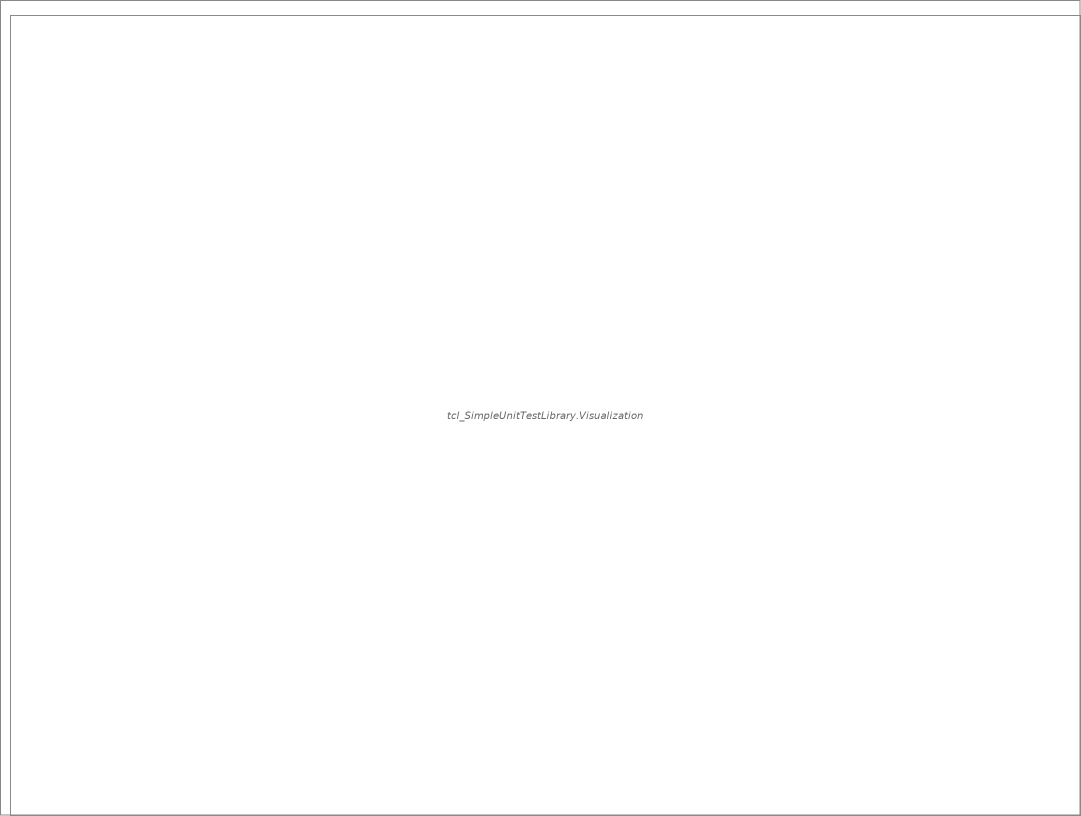
VISUALIZATION Visualization  // 1081x816
    Frame (10,15 1071x801)
        shows tcl_SimpleUnitTestLibrary.Visualization(TestRunner := PB_TestRunner.TestRunner)
END_VISUALIZATION

(* stored: Version 1.1.0.1, ProductVersion 3.1.4024.6
   Visu Visualization: Id {f7630f05-a200-0986-2471-7edcb76a9027} *)
